TYPE UDT 1271

TITLE =

VERSION : 0.1

  STRUCT

   Field : INT ;

  END_STRUCT ;

END_TYPE



FUNCTION_BLOCK FB 68

TITLE =

VERSION : 0.1

NAME : STD_DEVIATION

BEGIN

NETWORK

TITLE =

END_FUNCTION_BLOCK



FUNCTION FC 100 : VOID

TITLE =

VERSION : 0.1

BEGIN

NETWORK

TITLE =

END_FUNCTION



DATA_BLOCK DB 1

TITLE =

VERSION : 0.1

BEGIN

END_DATA_BLOCK



ORGANIZATION_BLOCK OB 1

TITLE =

VERSION : 0.1

BEGIN

NETWORK

TITLE =

END_ORGANIZATION_BLOCK

